(*********************************** G.D S.p.A. - Technical Department ***********************************
============= PROGRAM INFO ============
FOLDER:             TBD
MACHINES INVOLVED:  TBD 

============= DESCRIPTION =============
csp main interface program

============= REVISIONS ===============
Date		Version	 	Author      	Description             
----------	-------		------------  	--------------------------------------------
2019/09/27 	0000.00	 	M.Grasso		Creation of the PRG

**********************************************************************************************************)
PROGRAM _csp_transfer_crosspusher_low
VAR
END_VAR

;

END_PROGRAM

(* stored: Version 1.1.0.1, ProductVersion 3.1.4022.12
   POU _csp_transfer_crosspusher_low: Id {eea43640-4046-4c0f-8b86-f8c05e1b3959}, SpecialFunc None *)
